FUNCTION_BLOCK FB_WinchControl
VAR_INPUT
END_VAR
VAR_OUTPUT
END_VAR
VAR
END_VAR

END_FUNCTION_BLOCK

(* stored: Version 1.1.0.1, ProductVersion 3.1.4024.12
   POU FB_WinchControl: Id {afefc06e-bd78-485d-a26b-89efa2ded290}, SpecialFunc None *)
